FUNCTION_BLOCK FB_HighLevelSystem IMPLEMENTS ITF_HighLevelSystem
VAR_INPUT
END_VAR
VAR_OUTPUT
END_VAR
VAR
	fbSub : FB_Subsystem;
END_VAR

{warning 'Methodenimplementierung hinzufügen'}
METHOD PUBLIC doConditionCheck : eConditionCheck
END_METHOD

{warning 'Eigenschaftenimplementierung hinzufügen'}
PROPERTY PUBLIC eCondition : eConditionCheck
GET
END_GET
SET
END_SET
END_PROPERTY

{attribute 'monitoring' := 'variable'}
{attribute 'monitoring' := 'call'}
PROPERTY InputsFromOC : INT
SET
fbSub.Input := InputsFromOC;
END_SET
END_PROPERTY

{warning 'Eigenschaftenimplementierung hinzufügen'}
PROPERTY PUBLIC nErrorID : UDINT
GET
END_GET
SET
END_SET
END_PROPERTY

{attribute 'monitoring' := 'variable'}
{attribute 'monitoring' := 'call'}
PROPERTY OutputsToOC : INT
GET

OutputsToOC := fbSub.Output;
END_GET
END_PROPERTY

END_FUNCTION_BLOCK

(* stored: Version 1.1.0.1, ProductVersion 3.1.4024.12
   POU FB_HighLevelSystem: Id {abb331e1-7dbc-4c32-8e27-840e8b78c198}, SpecialFunc None
   Method doConditionCheck: Id {6411a928-d24d-49af-ab83-db46d4efcd4e}
   Property eCondition: Id {e500d94e-e145-43a5-8780-aad128ab23c5}
   Get Get: Id {aa4a8ad1-a4f2-4081-9627-73ab894a3755}
   Set Set: Id {7ed00226-229b-4e0f-8fa0-05d4f7c66428}
   Property InputsFromOC: Id {f1f52be5-7e43-4933-b235-803463f0b018}
   Set Set: Id {fd2b779b-3c69-49ac-b979-bfbf078e707e}
   Property nErrorID: Id {b4f21694-afab-4922-9136-ef2684b9a6cd}
   Get Get: Id {4d56beb3-4fe1-4603-9b5a-5da5f090d629}
   Set Set: Id {fb4871ec-5ac5-401a-9858-8bed394331b2}
   Property OutputsToOC: Id {663b89d4-3fa6-487d-9da8-5e7dc0db56dd}
   Get Get: Id {6c4b38f7-7261-4e78-a4c5-6213c217ee31} *)
